PROGRAM PRG_DPL_Z_EPS
VAR
    {attribute 'pytmc' := 'pv: CRIX:DPL:MMS:Z:EPS'}
    aDPL_Z_EPS 	    : ARRAY [1 .. 4] OF ST_EPSLimits;

    {attribute 'pytmc' := 'pv: CRIX:DPL:MMS:Z:EPS:OVRD_MODE'}
    bEPS_Override: BOOL := FALSE;
    {attribute 'pytmc' := 'pv: CRIX:DPL:MMS:Z:EPS:OVRD_COUNTDOWN'}
    tEPS_TimerCountDown : STRING := TIME_TO_STRING(T#0s);
    fbResetTimer : FB_RestTimer;

    bInit 		: BOOL := TRUE;
    bFullRange 	: BOOL;

    fbEPS		: FB_EPS;
    fbCheckEPS 	: FB_CheckEPS;
END_VAR

IF bInit THEN
    // Set Inital Values
    aDPL_Z_EPS[1].fBwd_Limits := -10;
    aDPL_Z_EPS[1].fFwd_Limits := 100;

    aDPL_Z_EPS[2].fBwd_Limits := 30;
    aDPL_Z_EPS[2].fFwd_Limits := 100;

    aDPL_Z_EPS[3].fBwd_Limits := 30;
    aDPL_Z_EPS[3].fFwd_Limits := 100;

    aDPL_Z_EPS[4].fBwd_Limits := 30;
    aDPL_Z_EPS[4].fFwd_Limits := 100;

    bInit := FALSE;
END_IF

fbEPS(eps:=aDPL_Z_EPS[2].stEPS);
fbEPS.setMessage('DPL X in [10, OBJ_X + 30]');
fbEPS.setBit(0, F_InRange(fDPL_X, 10, fOBJ_X + 30));

fbEPS(eps:=aDPL_Z_EPS[3].stEPS);
fbEPS.setMessage('RCC Y in [-34,10];RCC_Z in [-15,11]');
fbEPS.setBit(0, F_InRange(fRCC_Y, -34, 10));
fbEPS.setBit(1, F_InRange(fRCC_Z, -15, 11));

fbEPS(eps:=aDPL_Z_EPS[4].stEPS);
fbEPS.setMessage('RCC_Y in [-38,-34];RCC_Z in [-15,11];DPL_Y in [-1,40]');
fbEPS.setBit(0, F_InRange(fRCC_Y, -38, -34));
fbEPS.setBit(1, F_InRange(fRCC_Z, -15, 11));
fbEPS.setBit(2, F_InRange(fDPL_Y, -1, 40));

bFullRange := (NOT aDPL_Z_EPS[2].stEPS.bEPS_OK) AND (NOT aDPL_Z_EPS[3].stEPS.bEPS_OK) AND (NOT aDPL_Z_EPS[4].stEPS.bEPS_OK);

fbEPS(eps:=aDPL_Z_EPS[1].stEPS);
fbEPS.setMessage('Full Range');
fbEPS.setBit(0, bFullRange);

fbResetTimer(bInput:=bEPS_Override, tElapseTime:=tEPS_OVRD_RESET_TIME, tCountDown:=tEPS_TimerCountDown);
fbCheckEPS(stMotor:=M3, fPosition:=fDPL_Z, aEPSLimits:= aDPL_Z_EPS, stForwardMotorEPS:=M3.stEPSForwardEnable, stBackwardMotorEPS:= M3.stEPSBackwardEnable, bEPS_Override:=bEPS_Override);

END_PROGRAM

(* stored: Version 1.1.0.1, ProductVersion 3.1.4022.18
   POU PRG_DPL_Z_EPS: Id {2c285499-0d64-4304-a814-9959d7ef4cde}, SpecialFunc None *)
